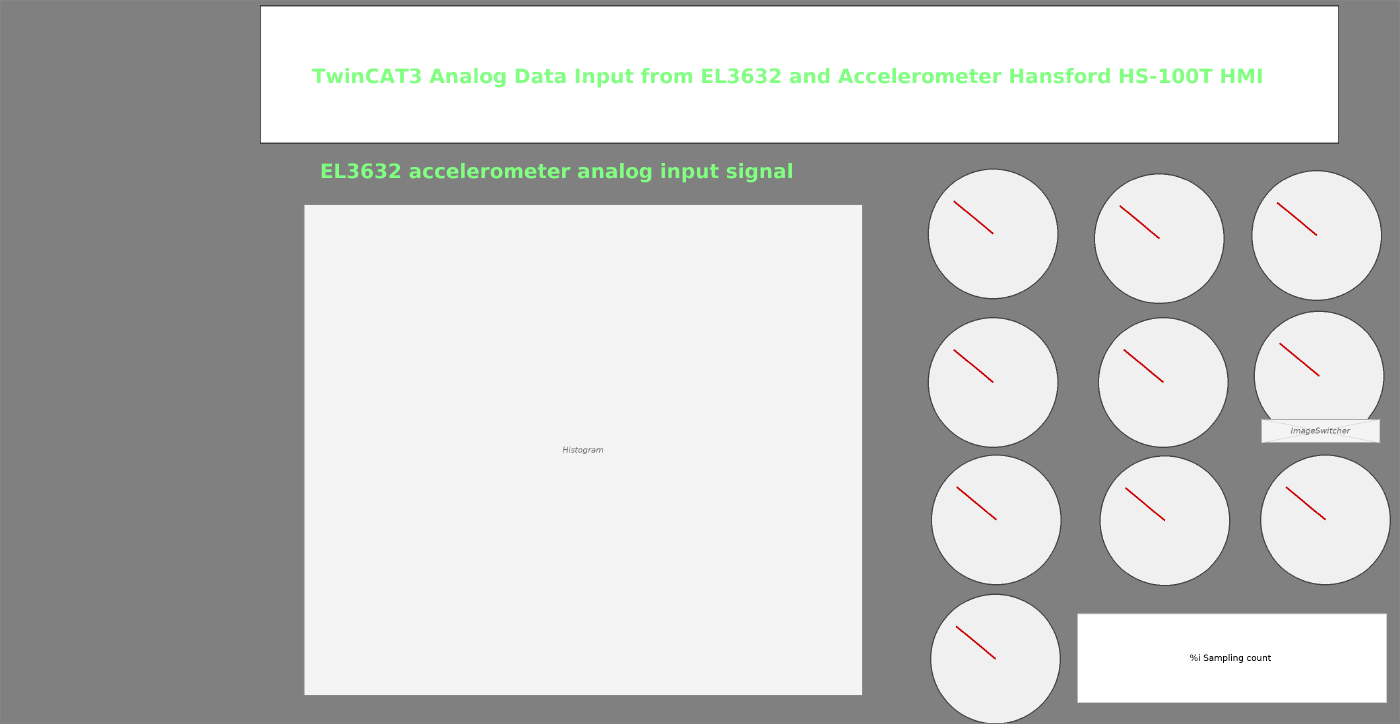
VISUALIZATION Visualization  // 1761x911, background image 
    Rectangle (327,7 1357x173)
    Label (417,155 575x120), "EL3632 accelerometer analog input signal"
    Textfield (1355,772 389x112), "%i Sampling count", text variable: MAIN.SAMPLE_COUNT_READ
    Meter360 (1155,212 188x164), value: MAIN.READ_DATA_1, style: Meter-Meter360-Gray, scale format: %.1f, scale 0..100
    Histogram (382,257 703x618), scale format: %.1f, scale -100..100
        p1518820177: MAIN.nAnalog
        p102497268: MAIN.nAnalog
        p788070771: ARRAY [1..10] OF INT
    Meter360 (1364,218 188x164), value: MAIN.READ_DATA_2, style: Meter-Meter360-Gray, scale format: %.1f, scale 0..100
    Meter360 (1562,214 188x164), value: MAIN.READ_DATA_3, style: Meter-Meter360-Gray, scale format: %.1f, scale 0..100
    Meter360 (1155,399 188x164), value: MAIN.READ_DATA_4, style: Meter-Meter360-Gray, scale format: %.1f, scale 0..100
    Meter360 (1369,399 188x164), value: MAIN.READ_DATA_5, style: Meter-Meter360-Gray, scale format: %.1f, scale 0..100
    Meter360 (1565,391 188x164), value: MAIN.READ_DATA_6, style: Meter-Meter360-Gray, scale format: %.1f, scale 0..100
    Meter360 (1159,572 188x164), value: MAIN.READ_DATA_7, style: Meter-Meter360-Gray, scale format: %.1f, scale 0..100
    Meter360 (1371,573 188x164), value: MAIN.READ_DATA_8, style: Meter-Meter360-Gray, scale format: %.1f, scale 0..100
    Meter360 (1573,572 188x164), value: MAIN.READ_DATA_9, style: Meter-Meter360-Gray, scale format: %.1f, scale 0..100
    Meter360 (1158,747 188x164), value: MAIN.READ_DATA_10, style: Meter-Meter360-Gray, scale format: %.1f, scale 0..100
    ImageSwitcher (1586,527 150x30), behaviour: TOGGLE
    Label (358,20 1266x151), "TwinCAT3 Analog Data Input from EL3632 and Accelerometer Hansford HS-100T HMI"
END_VISUALIZATION

(* stored: Version 1.1.0.1, ProductVersion 3.1.4024.16
   Visu Visualization: Id {5209e7c0-d504-401b-a552-d278f1762b3e} *)
